// Mitsubishi GX Works2 project: main   PLC: FX3U/FX3UC

PROGRAM MAIN
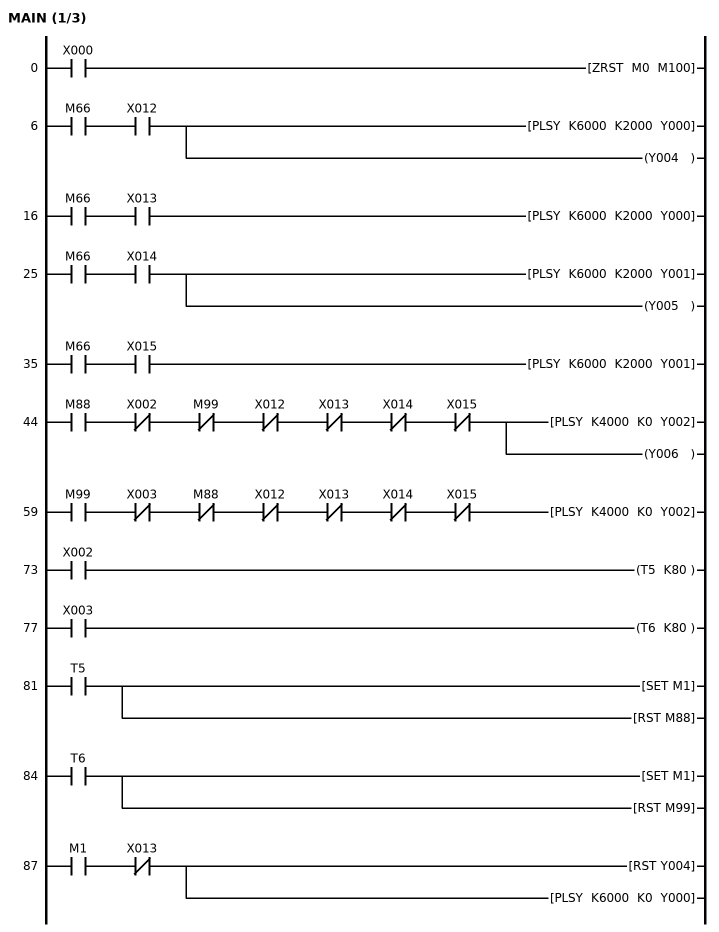
0     LD      X000
      ZRST    M0 M100
6     LD      M66
      AND     X012
      PLSY    K6000 K2000 Y000
      OUT     Y004
16    LD      M66
      AND     X013
      PLSY    K6000 K2000 Y000
25    LD      M66
      AND     X014
      PLSY    K6000 K2000 Y001
      OUT     Y005
35    LD      M66
      AND     X015
      PLSY    K6000 K2000 Y001
44    LD      M88
      ANI     X002
      ANI     M99
      ANI     X012
      ANI     X013
      ANI     X014
      ANI     X015
      PLSY    K4000 K0 Y002
      OUT     Y006
59    LD      M99
      ANI     X003
      ANI     M88
      ANI     X012
      ANI     X013
      ANI     X014
      ANI     X015
      PLSY    K4000 K0 Y002
73    LD      X002
      OUT     T5 K80
77    LD      X003
      OUT     T6 K80
81    LD      T5
      SET     M1
      RST     M88
84    LD      T6
      SET     M1
      RST     M99
87    LD      M1
      ANI     X013
      RST     Y004
      PLSY    K6000 K0 Y000
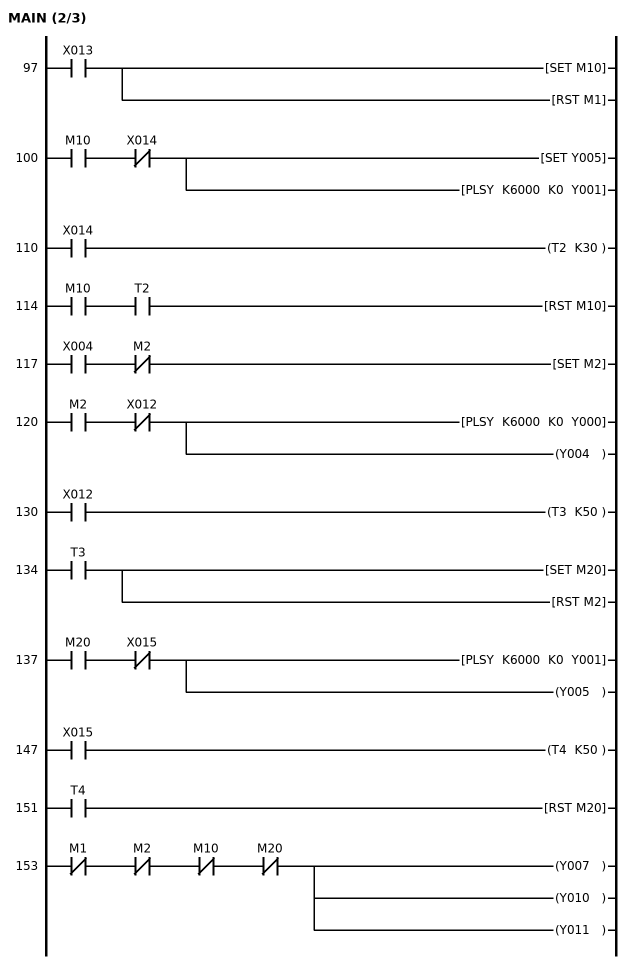
97    LD      X013
      SET     M10
      RST     M1
100   LD      M10
      ANI     X014
      SET     Y005
      PLSY    K6000 K0 Y001
110   LD      X014
      OUT     T2 K30
114   LD      M10
      AND     T2
      RST     M10
117   LD      X004
      ANI     M2
      SET     M2
120   LD      M2
      ANI     X012
      PLSY    K6000 K0 Y000
      OUT     Y004
130   LD      X012
      OUT     T3 K50
134   LD      T3
      SET     M20
      RST     M2
137   LD      M20
      ANI     X015
      PLSY    K6000 K0 Y001
      OUT     Y005
147   LD      X015
      OUT     T4 K50
151   LD      T4
      RST     M20
153   LDI     M1
      ANI     M2
      ANI     M10
      ANI     M20
      OUT     Y007
      OUT     Y010
      OUT     Y011
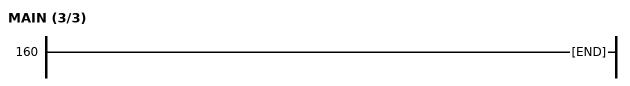
160   END
END_PROGRAM
